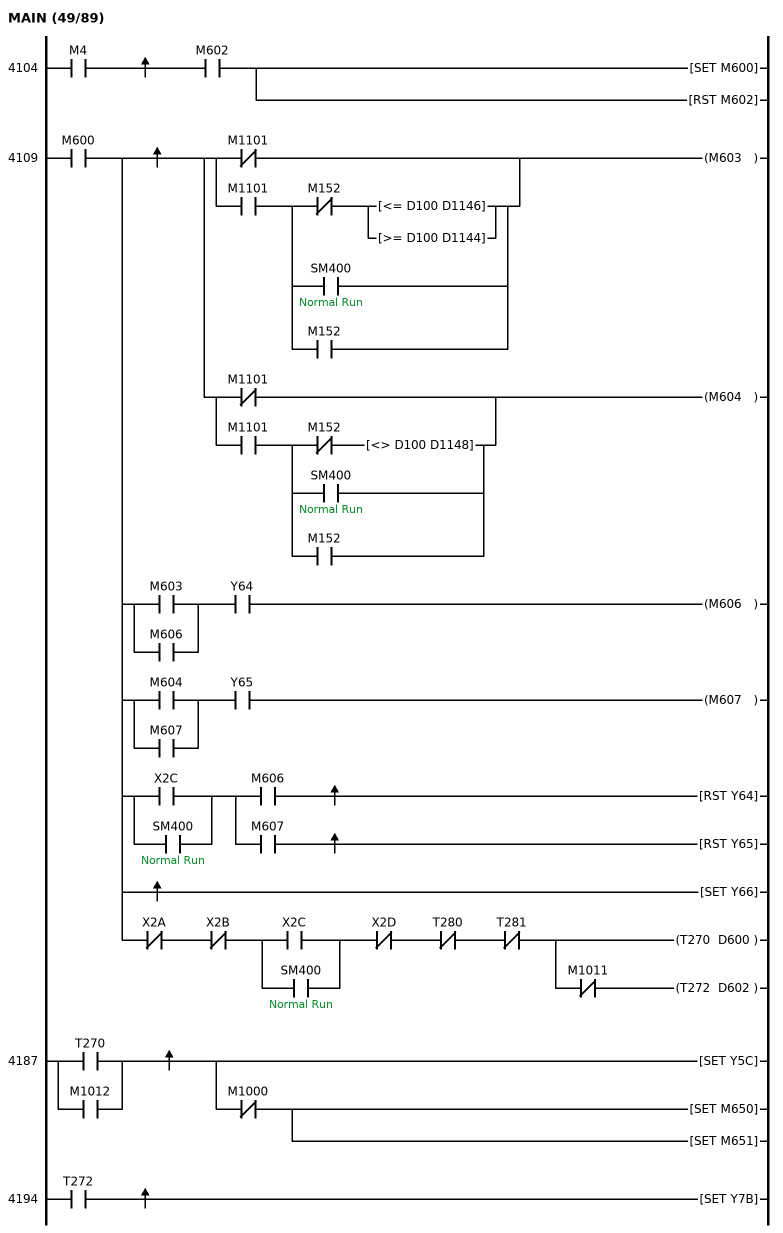
[picture p48: ladder of MAIN, rungs at steps 4104 to 4194]
4104  LD      M4
      MEP
      AND     M602
      SET     M600
      RST     M602
4109  LD      M600
      MPS
      MEP
      MPS
      LDI     M1101
      LD      M1101
      LDI     M152
      LD<=    D100 D1146
      OR>=    D100 D1144
      ANB
      OR      SM400  ; Normal Run
      OR      M152
      ANB
      ORB
      ANB
      OUT     M603
      MPP
      LDI     M1101
      LD      M1101
      LDI     M152
      AND<>   D100 D1148
      OR      SM400  ; Normal Run
      OR      M152
      ANB
      ORB
      ANB
      OUT     M604
      MRD
      LD      M603
      OR      M606
      ANB
      AND     Y64
      OUT     M606
      MRD
      LD      M604
      OR      M607
      ANB
      AND     Y65
      OUT     M607
      MRD
      LD      X2C
      OR      SM400  ; Normal Run
      ANB
      MPS
      AND     M606
      MEP
      RST     Y64
      MPP
      AND     M607
      MEP
      RST     Y65
      MRD
      MEP
      SET     Y66
      MPP
      ANI     X2A
      ANI     X2B
      LD      X2C
      OR      SM400  ; Normal Run
      ANB
      ANI     X2D
      ANI     T280
      ANI     T281
      OUT     T270 D600
      ANI     M1011
      OUT     T272 D602
4187  LD      T270
      OR      M1012
      MEP
      SET     Y5C
      ANI     M1000
      SET     M650
      SET     M651
4194  LD      T272
      MEP
      SET     Y7B
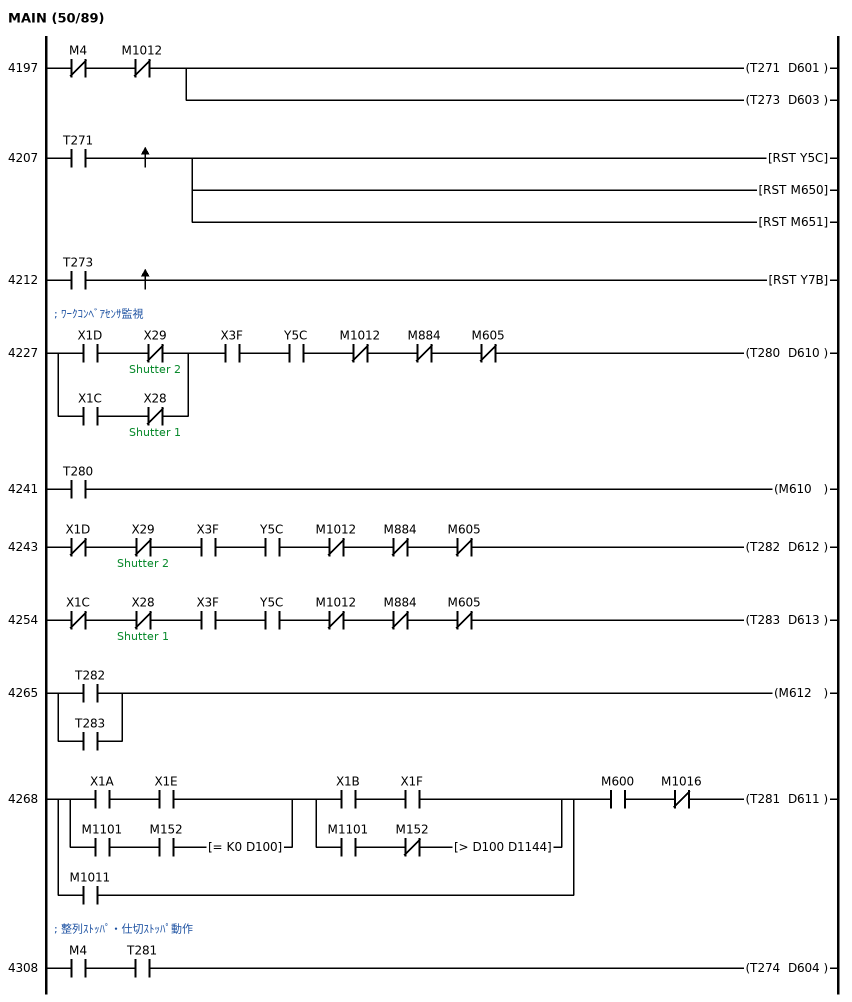
4197  LDI     M4
      ANI     M1012
      OUT     T271 D601
      OUT     T273 D603
4207  LD      T271
      MEP
      RST     Y5C
      RST     M650
      RST     M651
4212  LD      T273
      MEP
      RST     Y7B
; ﾜｰｸｺﾝﾍﾞｱｾﾝｻ監視
4227  LD      X1D
      ANI     X29  ; Shutter 2
      LD      X1C
      ANI     X28  ; Shutter 1
      ORB
      AND     X3F
      AND     Y5C
      ANI     M1012
      ANI     M884
      ANI     M605
      OUT     T280 D610
4241  LD      T280
      OUT     M610
4243  LDI     X1D
      ANI     X29  ; Shutter 2
      AND     X3F
      AND     Y5C
      ANI     M1012
      ANI     M884
      ANI     M605
      OUT     T282 D612
4254  LDI     X1C
      ANI     X28  ; Shutter 1
      AND     X3F
      AND     Y5C
      ANI     M1012
      ANI     M884
      ANI     M605
      OUT     T283 D613
4265  LD      T282
      OR      T283
      OUT     M612
4268  LD      X1A
      AND     X1E
      LD      M1101
      AND     M152
      AND=    K0 D100
      ORB
      LD      X1B
      AND     X1F
      LD      M1101
      ANI     M152
      AND>    D100 D1144
      ORB
      ANB
      OR      M1011
      AND     M600
      ANI     M1016
      OUT     T281 D611
; 整列ｽﾄｯﾊﾟ・仕切ｽﾄｯﾊﾟ動作
4308  LD      M4
      AND     T281
      OUT     T274 D604
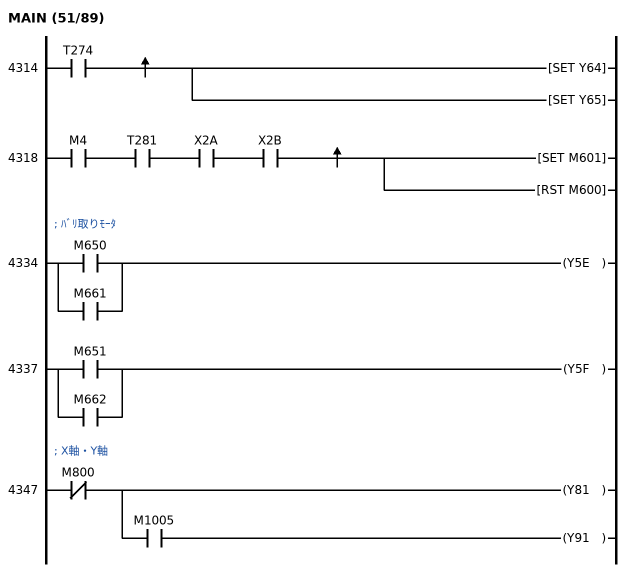
4314  LD      T274
      MEP
      SET     Y64
      SET     Y65
4318  LD      M4
      AND     T281
      AND     X2A
      AND     X2B
      MEP
      SET     M601
      RST     M600
; ﾊﾞﾘ取りﾓｰﾀ
4334  LD      M650
      OR      M661
      OUT     Y5E
4337  LD      M651
      OR      M662
      OUT     Y5F
; X軸・Y軸
; 
4347  LDI     M800
      OUT     Y81
      AND     M1005
      OUT     Y91
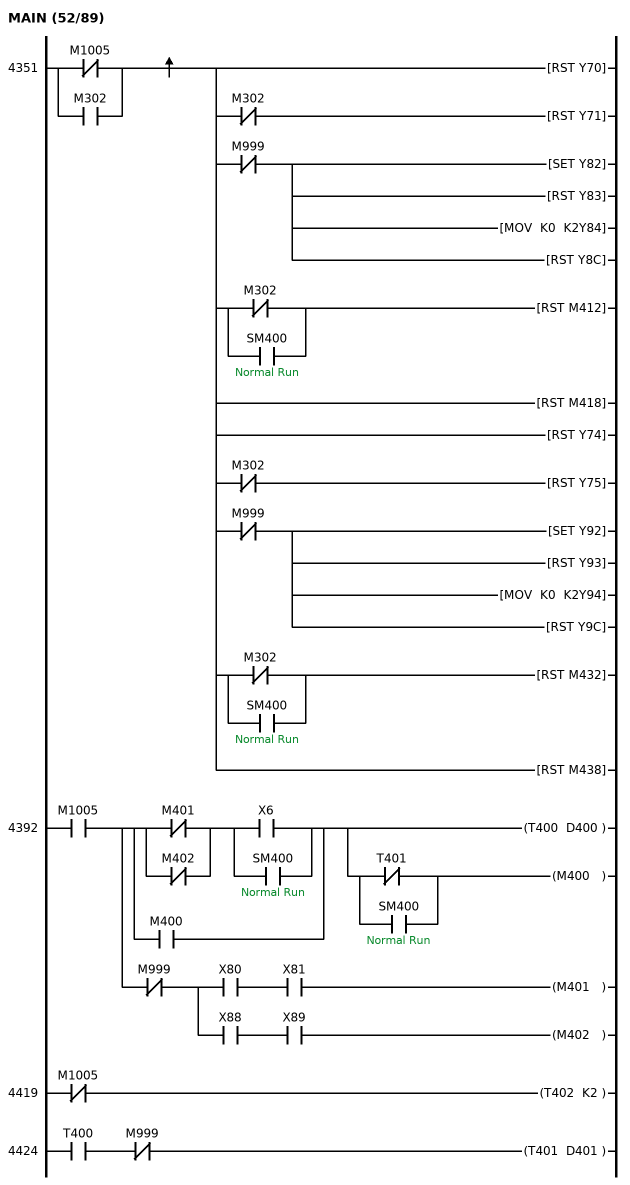
4351  LDI     M1005
      OR      M302
      MEP
      RST     Y70
      MPS
      ANI     M302
      RST     Y71
      MRD
      ANI     M999
      SET     Y82
      RST     Y83
      MOV     K0 K2Y84
      RST     Y8C
      MRD
      LDI     M302
      OR      SM400  ; Normal Run
      ANB
      RST     M412
      MPP
      RST     M418
      RST     Y74
      MPS
      ANI     M302
      RST     Y75
      MRD
      ANI     M999
      SET     Y92
      RST     Y93
      MOV     K0 K2Y94
      RST     Y9C
      MRD
      LDI     M302
      OR      SM400  ; Normal Run
      ANB
      RST     M432
      MPP
      RST     M438
4392  LD      M1005
      MPS
      LDI     M401
      ORI     M402
      LD      X6
      OR      SM400  ; Normal Run
      ANB
      OR      M400
      ANB
      OUT     T400 D400
      LDI     T401
      OR      SM400  ; Normal Run
      ANB
      OUT     M400
      MPP
      ANI     M999
      MPS
      AND     X80
      AND     X81
      OUT     M401
      MPP
      AND     X88
      AND     X89
      OUT     M402
4419  LDI     M1005
      OUT     T402 K2
4424  LD      T400
      ANI     M999
      OUT     T401 D401
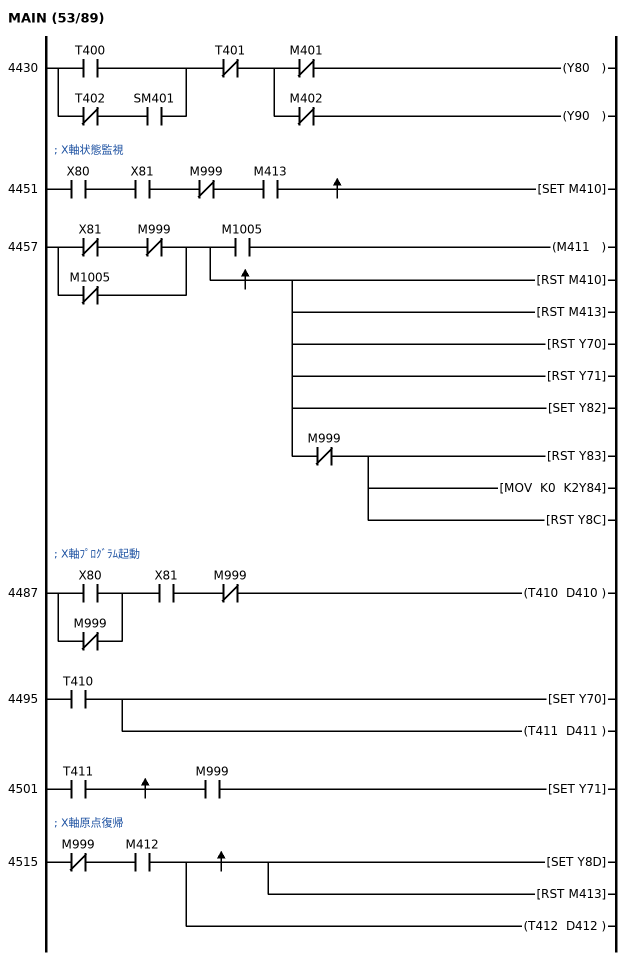
4430  LD      T400
      LDI     T402
      AND     SM401
      ORB
      ANI     T401
      MPS
      ANI     M401
      OUT     Y80
      MPP
      ANI     M402
      OUT     Y90
; X軸状態監視
4451  LD      X80
      AND     X81
      ANI     M999
      AND     M413
      MEP
      SET     M410
4457  LDI     X81
      ANI     M999
      ORI     M1005
      MPS
      AND     M1005
      OUT     M411
      MPP
      MEP
      RST     M410
      RST     M413
      RST     Y70
      RST     Y71
      SET     Y82
      ANI     M999
      RST     Y83
      MOV     K0 K2Y84
      RST     Y8C
; X軸ﾌﾟﾛｸﾞﾗﾑ起動
4487  LD      X80
      ORI     M999
      AND     X81
      ANI     M999
      OUT     T410 D410
4495  LD      T410
      SET     Y70
      OUT     T411 D411
4501  LD      T411
      MEP
      AND     M999
      SET     Y71
; X軸原点復帰
4515  LDI     M999
      AND     M412
      MPS
      MEP
      SET     Y8D
      RST     M413
      MPP
      OUT     T412 D412
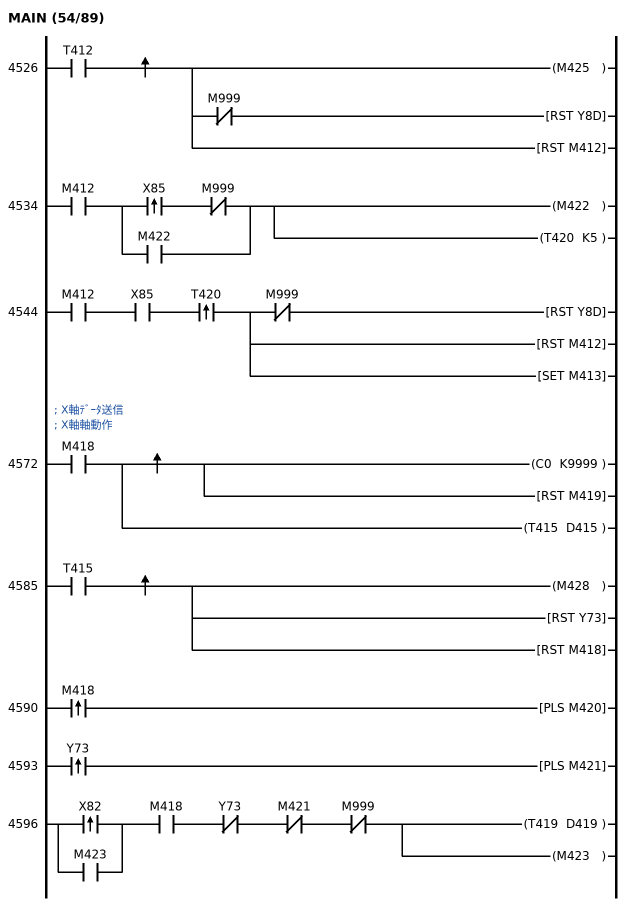
4526  LD      T412
      MEP
      OUT     M425
      MPS
      ANI     M999
      RST     Y8D
      MPP
      RST     M412
4534  LD      M412
      LDP     X85
      ANI     M999
      OR      M422
      ANB
      OUT     M422
      OUT     T420 K5
4544  LD      M412
      AND     X85
      ANDP    T420
      MPS
      ANI     M999
      RST     Y8D
      MPP
      RST     M412
      SET     M413
; X軸ﾃﾞｰﾀ送信
; X軸軸動作
4572  LD      M418
      MPS
      MEP
      OUT     C0 K9999
      RST     M419
      MPP
      OUT     T415 D415
4585  LD      T415
      MEP
      OUT     M428
      RST     Y73
      RST     M418
4590  LDP     M418
      PLS     M420
4593  LDP     Y73
      PLS     M421
4596  LDP     X82
      OR      M423
      AND     M418
      ANI     Y73
      ANI     M421
      ANI     M999
      OUT     T419 D419
      OUT     M423
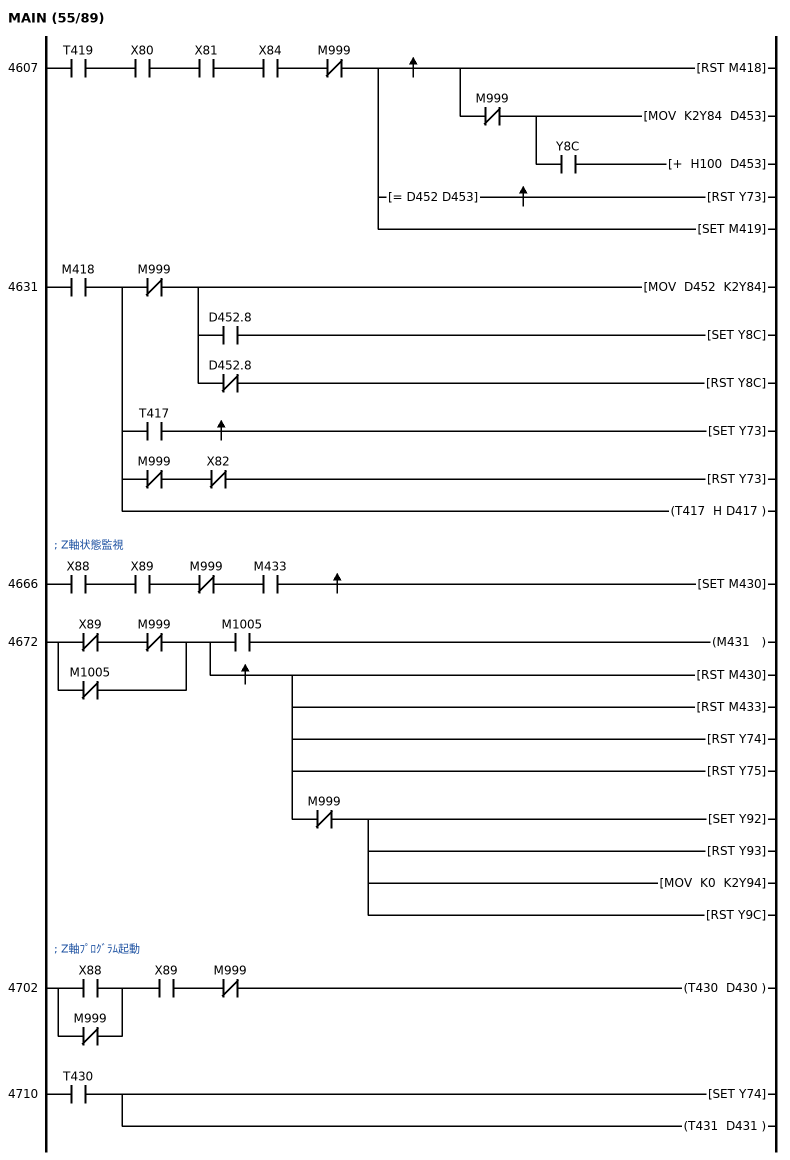
4607  LD      T419
      AND     X80
      AND     X81
      AND     X84
      ANI     M999
      MPS
      MEP
      RST     M418
      ANI     M999
      MOV     K2Y84 D453
      AND     Y8C
      +       H100 D453
      MRD
      AND=    D452 D453
      MEP
      RST     Y73
      MPP
      SET     M419
4631  LD      M418
      MPS
      ANI     M999
      MOV     D452 K2Y84
      MPS
      AND     D452.8
      SET     Y8C
      MPP
      ANI     D452.8
      RST     Y8C
      MRD
      AND     T417
      MEP
      SET     Y73
      MRD
      ANI     M999
      ANI     X82
      RST     Y73
      MPP
      OUTH    T417 D417
; Z軸状態監視
4666  LD      X88
      AND     X89
      ANI     M999
      AND     M433
      MEP
      SET     M430
4672  LDI     X89
      ANI     M999
      ORI     M1005
      MPS
      AND     M1005
      OUT     M431
      MPP
      MEP
      RST     M430
      RST     M433
      RST     Y74
      RST     Y75
      ANI     M999
      SET     Y92
      RST     Y93
      MOV     K0 K2Y94
      RST     Y9C
; Z軸ﾌﾟﾛｸﾞﾗﾑ起動
4702  LD      X88
      ORI     M999
      AND     X89
      ANI     M999
      OUT     T430 D430
4710  LD      T430
      SET     Y74
      OUT     T431 D431
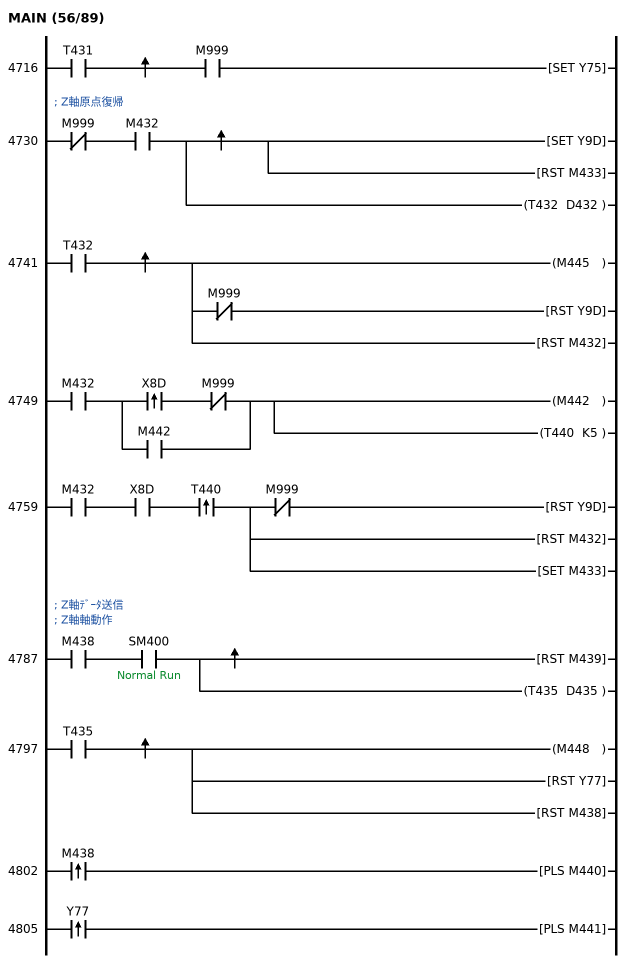
4716  LD      T431
      MEP
      AND     M999
      SET     Y75
; Z軸原点復帰
4730  LDI     M999
      AND     M432
      MPS
      MEP
      SET     Y9D
      RST     M433
      MPP
      OUT     T432 D432
4741  LD      T432
      MEP
      OUT     M445
      MPS
      ANI     M999
      RST     Y9D
      MPP
      RST     M432
4749  LD      M432
      LDP     X8D
      ANI     M999
      OR      M442
      ANB
      OUT     M442
      OUT     T440 K5
4759  LD      M432
      AND     X8D
      ANDP    T440
      MPS
      ANI     M999
      RST     Y9D
      MPP
      RST     M432
      SET     M433
; Z軸ﾃﾞｰﾀ送信
; Z軸軸動作
4787  LD      M438
      AND     SM400  ; Normal Run
      MPS
      MEP
      RST     M439
      MPP
      OUT     T435 D435
4797  LD      T435
      MEP
      OUT     M448
      RST     Y77
      RST     M438
4802  LDP     M438
      PLS     M440
4805  LDP     Y77
      PLS     M441
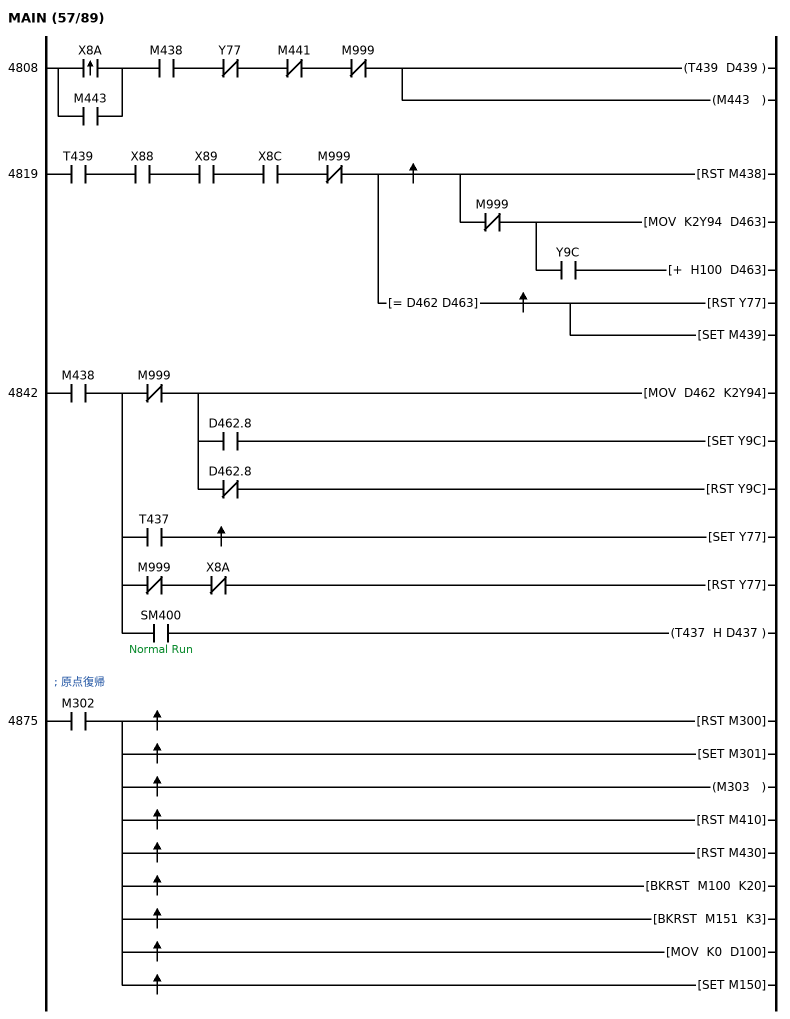
4808  LDP     X8A
      OR      M443
      AND     M438
      ANI     Y77
      ANI     M441
      ANI     M999
      OUT     T439 D439
      OUT     M443
4819  LD      T439
      AND     X88
      AND     X89
      AND     X8C
      ANI     M999
      MPS
      MEP
      RST     M438
      ANI     M999
      MOV     K2Y94 D463
      AND     Y9C
      +       H100 D463
      MPP
      AND=    D462 D463
      MEP
      RST     Y77
      SET     M439
4842  LD      M438
      MPS
      ANI     M999
      MOV     D462 K2Y94
      MPS
      AND     D462.8
      SET     Y9C
      MPP
      ANI     D462.8
      RST     Y9C
      MRD
      AND     T437
      MEP
      SET     Y77
      MRD
      ANI     M999
      ANI     X8A
      RST     Y77
      MPP
      AND     SM400  ; Normal Run
      OUTH    T437 D437
; 原点復帰
; 
4875  LD      M302
      MPS
      MEP
      RST     M300
      MRD
      MEP
      SET     M301
      MRD
      MEP
      OUT     M303
      MRD
      MEP
      RST     M410
      MRD
      MEP
      RST     M430
      MRD
      MEP
      BKRST   M100 K20
      MRD
      MEP
      BKRST   M151 K3
      MRD
      MEP
      MOV     K0 D100
      MPP
      MEP
      SET     M150
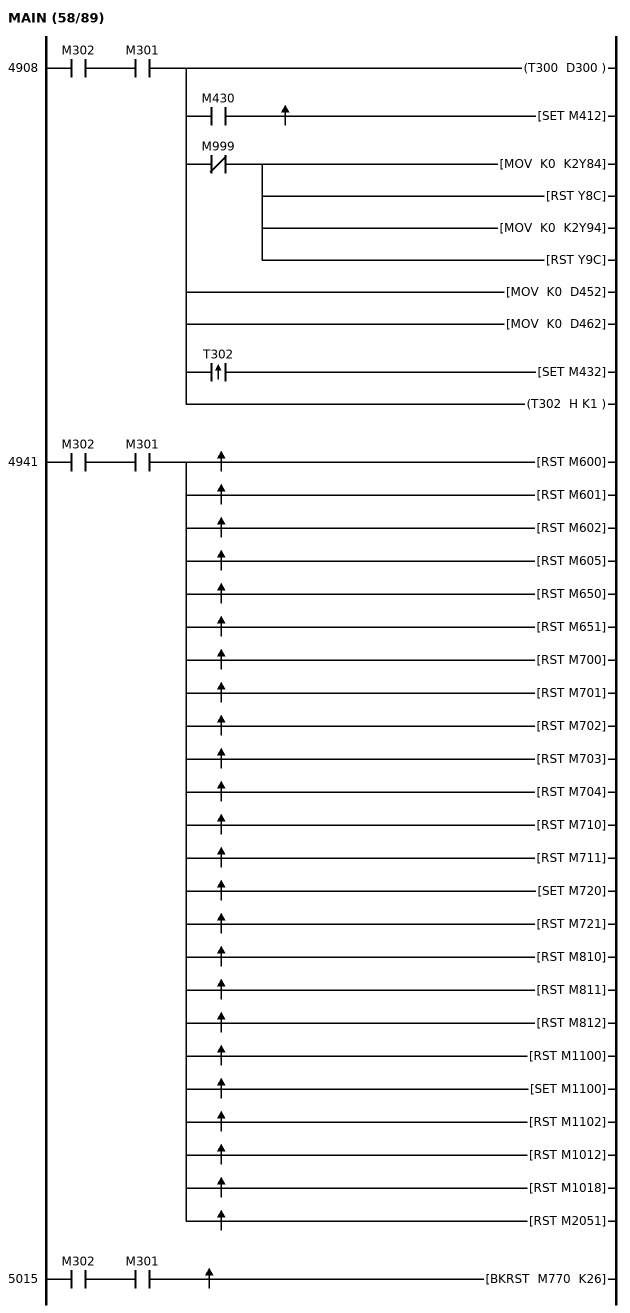
4908  LD      M302
      AND     M301
      OUT     T300 D300
      MPS
      AND     M430
      MEP
      SET     M412
      MRD
      ANI     M999
      MOV     K0 K2Y84
      RST     Y8C
      MOV     K0 K2Y94
      RST     Y9C
      MPP
      MOV     K0 D452
      MOV     K0 D462
      MPS
      ANDP    T302
      SET     M432
      MPP
      OUTH    T302 K1
4941  LD      M302
      AND     M301
      MPS
      MEP
      RST     M600
      MRD
      MEP
      RST     M601
      MRD
      MEP
      RST     M602
      MRD
      MEP
      RST     M605
      MRD
      MEP
      RST     M650
      MRD
      MEP
      RST     M651
      MRD
      MEP
      RST     M700
      MRD
      MEP
      RST     M701
      MRD
      MEP
      RST     M702
      MRD
      MEP
      RST     M703
      MRD
      MEP
      RST     M704
      MRD
      MEP
      RST     M710
      MRD
      MEP
      RST     M711
      MRD
      MEP
      SET     M720
      MRD
      MEP
      RST     M721
      MRD
      MEP
      RST     M810
      MRD
      MEP
      RST     M811
      MRD
      MEP
      RST     M812
      MRD
      MEP
      RST     M1100
      MRD
      MEP
      SET     M1100
      MRD
      MEP
      RST     M1102
      MRD
      MEP
      RST     M1012
      MRD
      MEP
      RST     M1018
      MPP
      MEP
      RST     M2051
5015  LD      M302
      AND     M301
      MEP
      BKRST   M770 K26
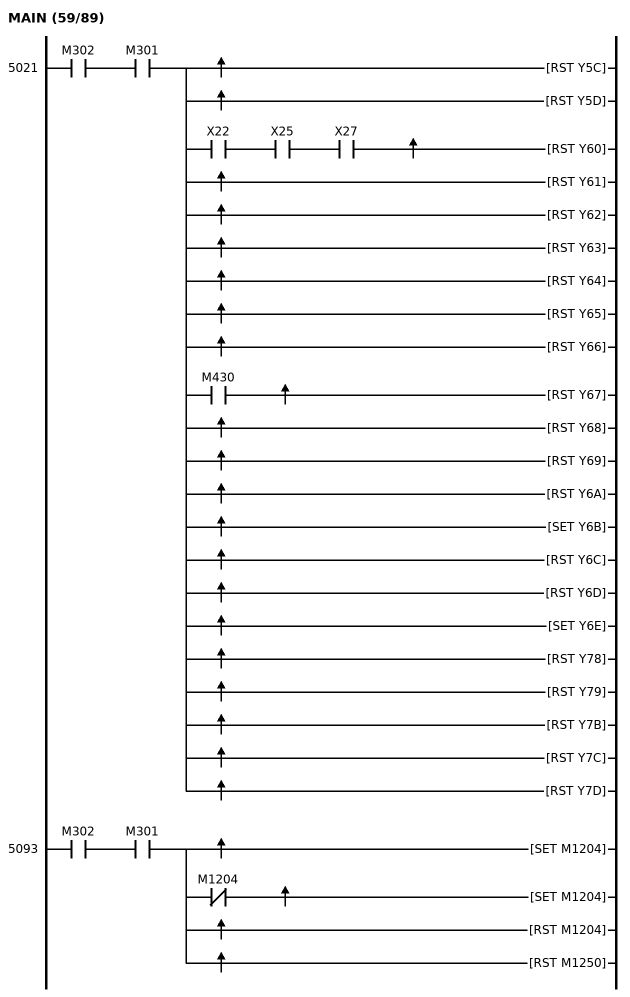
5021  LD      M302
      AND     M301
      MPS
      MEP
      RST     Y5C
      MRD
      MEP
      RST     Y5D
      MRD
      AND     X22
      AND     X25
      AND     X27
      MEP
      RST     Y60
      MRD
      MEP
      RST     Y61
      MRD
      MEP
      RST     Y62
      MRD
      MEP
      RST     Y63
      MRD
      MEP
      RST     Y64
      MRD
      MEP
      RST     Y65
      MRD
      MEP
      RST     Y66
      MRD
      AND     M430
      MEP
      RST     Y67
      MRD
      MEP
      RST     Y68
      MRD
      MEP
      RST     Y69
      MRD
      MEP
      RST     Y6A
      MRD
      MEP
      SET     Y6B
      MRD
      MEP
      RST     Y6C
      MRD
      MEP
      RST     Y6D
      MRD
      MEP
      SET     Y6E
      MRD
      MEP
      RST     Y78
      MRD
      MEP
      RST     Y79
      MRD
      MEP
      RST     Y7B
      MRD
      MEP
      RST     Y7C
      MPP
      MEP
      RST     Y7D
5093  LD      M302
      AND     M301
      MPS
      MEP
      SET     M1204
      MRD
      ANI     M1204
      MEP
      SET     M1204
      MRD
      MEP
      RST     M1204
      MPP
      MEP
      RST     M1250
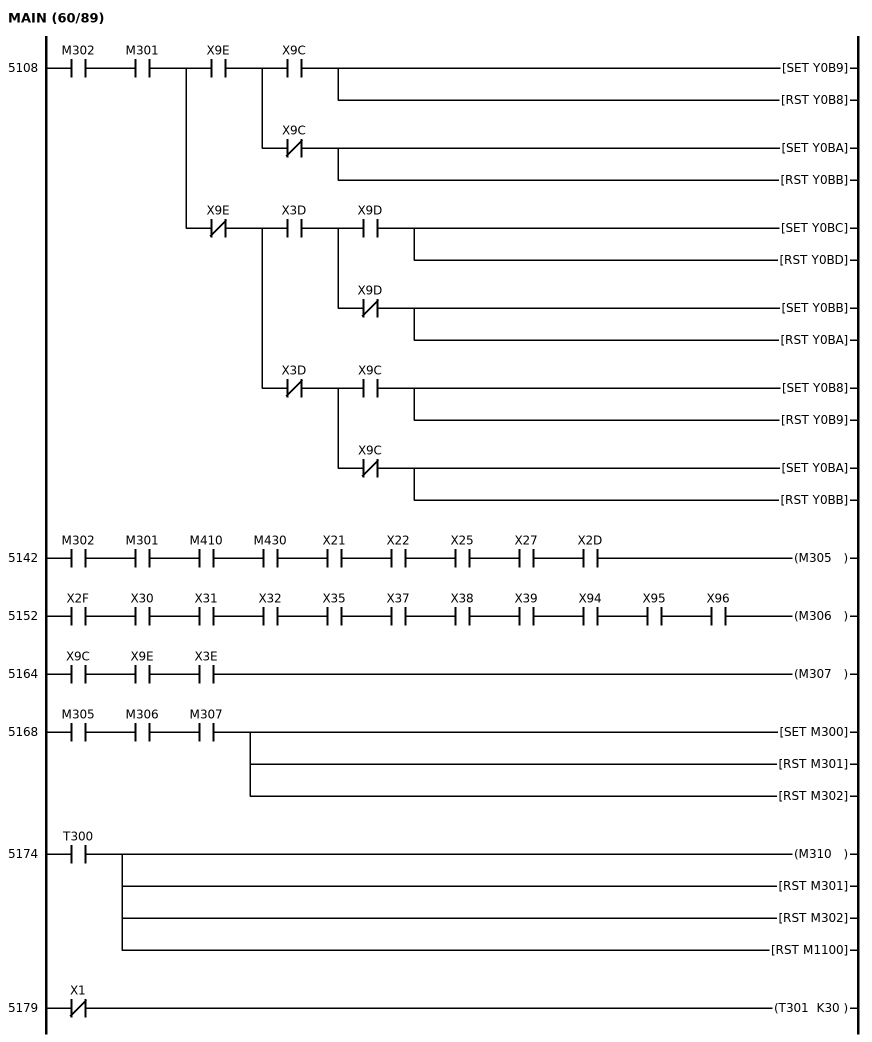
5108  LD      M302
      AND     M301
      MPS
      AND     X9E
      MPS
      AND     X9C
      SET     Y0B9
      RST     Y0B8
      MPP
      ANI     X9C
      SET     Y0BA
      RST     Y0BB
      MPP
      ANI     X9E
      MPS
      AND     X3D
      MPS
      AND     X9D
      SET     Y0BC
      RST     Y0BD
      MPP
      ANI     X9D
      SET     Y0BB
      RST     Y0BA
      MPP
      ANI     X3D
      MPS
      AND     X9C
      SET     Y0B8
      RST     Y0B9
      MPP
      ANI     X9C
      SET     Y0BA
      RST     Y0BB
5142  LD      M302
      AND     M301
      AND     M410
      AND     M430
      AND     X21
      AND     X22
      AND     X25
      AND     X27
      AND     X2D
      OUT     M305
5152  LD      X2F
      AND     X30
      AND     X31
      AND     X32
      AND     X35
      AND     X37
      AND     X38
      AND     X39
      AND     X94
      AND     X95
      AND     X96
      OUT     M306
5164  LD      X9C
      AND     X9E
      AND     X3E
      OUT     M307
5168  LD      M305
      AND     M306
      AND     M307
      SET     M300
      RST     M301
      RST     M302
5174  LD      T300
      OUT     M310
      RST     M301
      RST     M302
      RST     M1100
5179  LDI     X1
      OUT     T301 K30
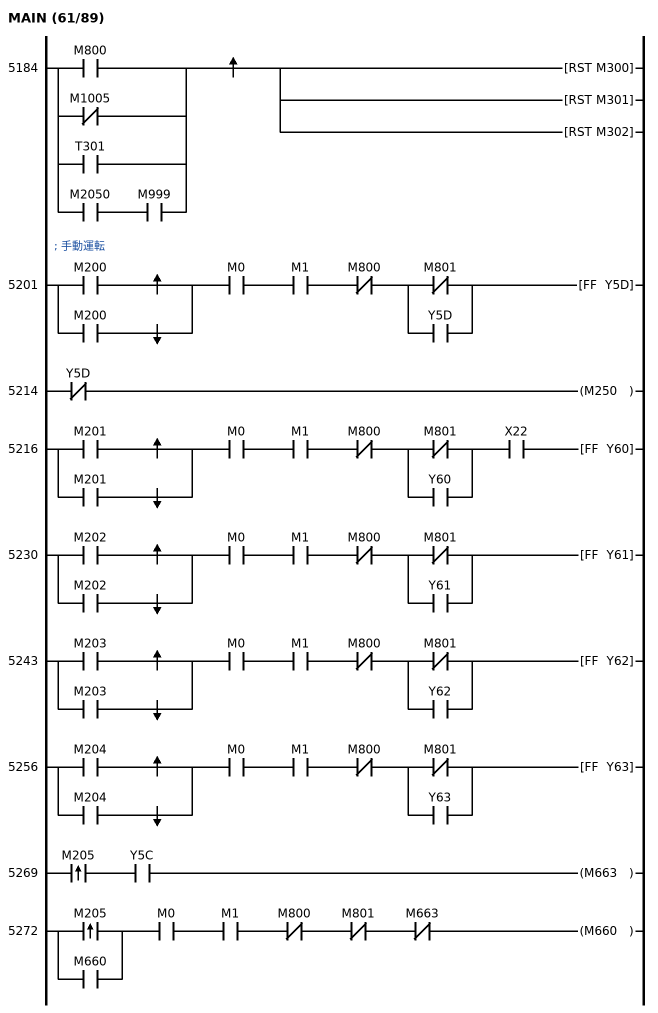
5184  LD      M800
      ORI     M1005
      OR      T301
      LD      M2050
      AND     M999
      ORB
      MEP
      RST     M300
      RST     M301
      RST     M302
; 手動運転
; 
5201  LD      M200
      MEP
      LD      M200
      MEF
      ORB
      AND     M0
      AND     M1
      ANI     M800
      LDI     M801
      OR      Y5D
      ANB
      FF      Y5D
5214  LDI     Y5D
      OUT     M250
5216  LD      M201
      MEP
      LD      M201
      MEF
      ORB
      AND     M0
      AND     M1
      ANI     M800
      LDI     M801
      OR      Y60
      ANB
      AND     X22
      FF      Y60
5230  LD      M202
      MEP
      LD      M202
      MEF
      ORB
      AND     M0
      AND     M1
      ANI     M800
      LDI     M801
      OR      Y61
      ANB
      FF      Y61
5243  LD      M203
      MEP
      LD      M203
      MEF
      ORB
      AND     M0
      AND     M1
      ANI     M800
      LDI     M801
      OR      Y62
      ANB
      FF      Y62
5256  LD      M204
      MEP
      LD      M204
      MEF
      ORB
      AND     M0
      AND     M1
      ANI     M800
      LDI     M801
      OR      Y63
      ANB
      FF      Y63
5269  LDP     M205
      AND     Y5C
      OUT     M663
5272  LDP     M205
      OR      M660
      AND     M0
      AND     M1
      ANI     M800
      ANI     M801
      ANI     M663
      OUT     M660
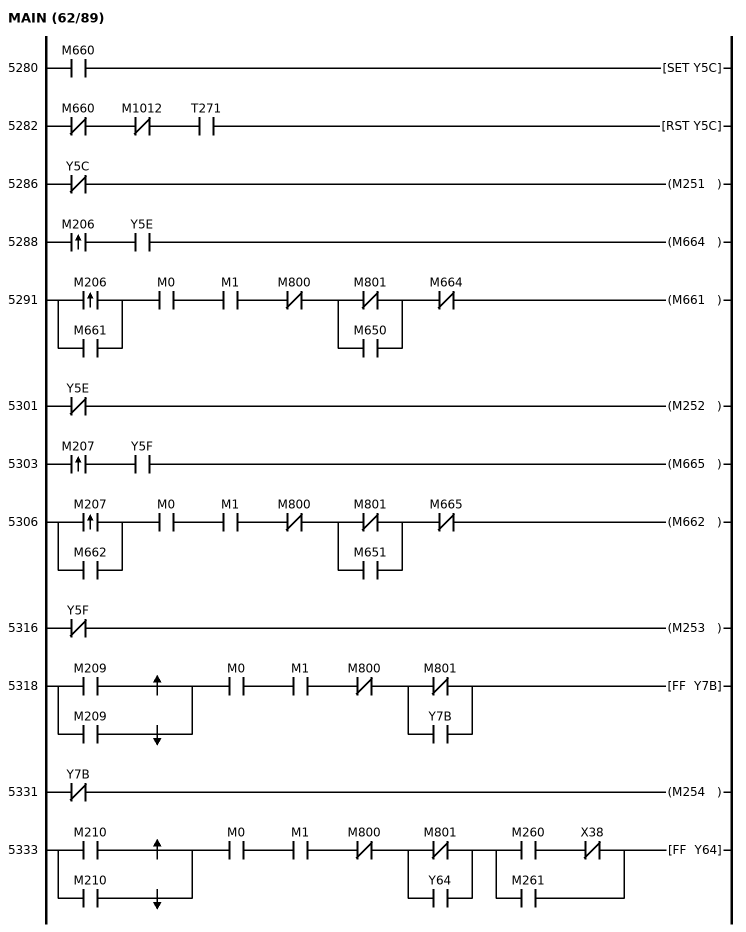
5280  LD      M660
      SET     Y5C
5282  LDI     M660
      ANI     M1012
      AND     T271
      RST     Y5C
5286  LDI     Y5C
      OUT     M251
5288  LDP     M206
      AND     Y5E
      OUT     M664
5291  LDP     M206
      OR      M661
      AND     M0
      AND     M1
      ANI     M800
      LDI     M801
      OR      M650
      ANB
      ANI     M664
      OUT     M661
5301  LDI     Y5E
      OUT     M252
5303  LDP     M207
      AND     Y5F
      OUT     M665
5306  LDP     M207
      OR      M662
      AND     M0
      AND     M1
      ANI     M800
      LDI     M801
      OR      M651
      ANB
      ANI     M665
      OUT     M662
5316  LDI     Y5F
      OUT     M253
5318  LD      M209
      MEP
      LD      M209
      MEF
      ORB
      AND     M0
      AND     M1
      ANI     M800
      LDI     M801
      OR      Y7B
      ANB
      FF      Y7B
5331  LDI     Y7B
      OUT     M254
5333  LD      M210
      MEP
      LD      M210
      MEF
      ORB
      AND     M0
      AND     M1
      ANI     M800
      LDI     M801
      OR      Y64
      ANB
      LD      M260
      ANI     X38
      OR      M261
      ANB
      FF      Y64
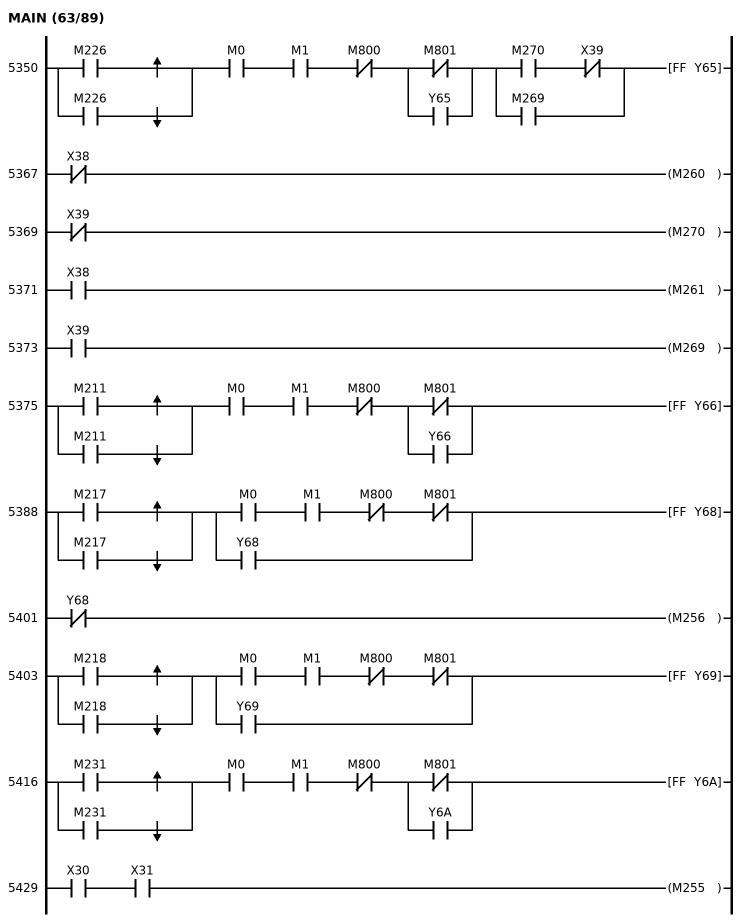
5350  LD      M226
      MEP
      LD      M226
      MEF
      ORB
      AND     M0
      AND     M1
      ANI     M800
      LDI     M801
      OR      Y65
      ANB
      LD      M270
      ANI     X39
      OR      M269
      ANB
      FF      Y65
5367  LDI     X38
      OUT     M260
5369  LDI     X39
      OUT     M270
5371  LD      X38
      OUT     M261
5373  LD      X39
      OUT     M269
5375  LD      M211
      MEP
      LD      M211
      MEF
      ORB
      AND     M0
      AND     M1
      ANI     M800
      LDI     M801
      OR      Y66
      ANB
      FF      Y66
5388  LD      M217
      MEP
      LD      M217
      MEF
      ORB
      LD      M0
      AND     M1
      ANI     M800
      ANI     M801
      OR      Y68
      ANB
      FF      Y68
5401  LDI     Y68
      OUT     M256
5403  LD      M218
      MEP
      LD      M218
      MEF
      ORB
      LD      M0
      AND     M1
      ANI     M800
      ANI     M801
      OR      Y69
      ANB
      FF      Y69
5416  LD      M231
      MEP
      LD      M231
      MEF
      ORB
      AND     M0
      AND     M1
      ANI     M800
      LDI     M801
      OR      Y6A
      ANB
      FF      Y6A
5429  LD      X30
      AND     X31
      OUT     M255
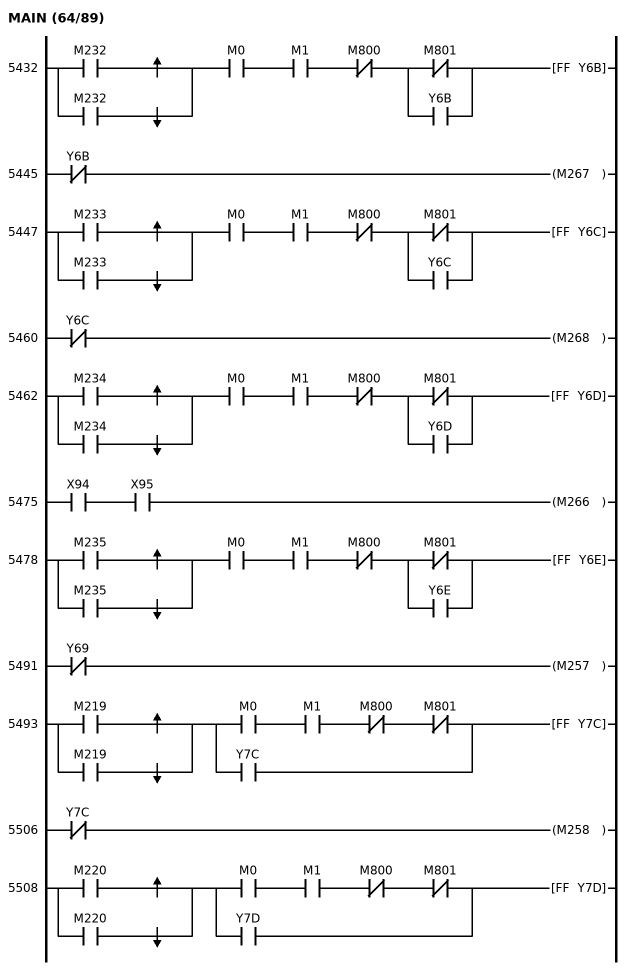
5432  LD      M232
      MEP
      LD      M232
      MEF
      ORB
      AND     M0
      AND     M1
      ANI     M800
      LDI     M801
      OR      Y6B
      ANB
      FF      Y6B
5445  LDI     Y6B
      OUT     M267
5447  LD      M233
      MEP
      LD      M233
      MEF
      ORB
      AND     M0
      AND     M1
      ANI     M800
      LDI     M801
      OR      Y6C
      ANB
      FF      Y6C
5460  LDI     Y6C
      OUT     M268
5462  LD      M234
      MEP
      LD      M234
      MEF
      ORB
      AND     M0
      AND     M1
      ANI     M800
      LDI     M801
      OR      Y6D
      ANB
      FF      Y6D
5475  LD      X94
      AND     X95
      OUT     M266
5478  LD      M235
      MEP
      LD      M235
      MEF
      ORB
      AND     M0
      AND     M1
      ANI     M800
      LDI     M801
      OR      Y6E
      ANB
      FF      Y6E
5491  LDI     Y69
      OUT     M257
5493  LD      M219
      MEP
      LD      M219
      MEF
      ORB
      LD      M0
      AND     M1
      ANI     M800
      ANI     M801
      OR      Y7C
      ANB
      FF      Y7C
5506  LDI     Y7C
      OUT     M258
5508  LD      M220
      MEP
      LD      M220
      MEF
      ORB
      LD      M0
      AND     M1
      ANI     M800
      ANI     M801
      OR      Y7D
      ANB
      FF      Y7D
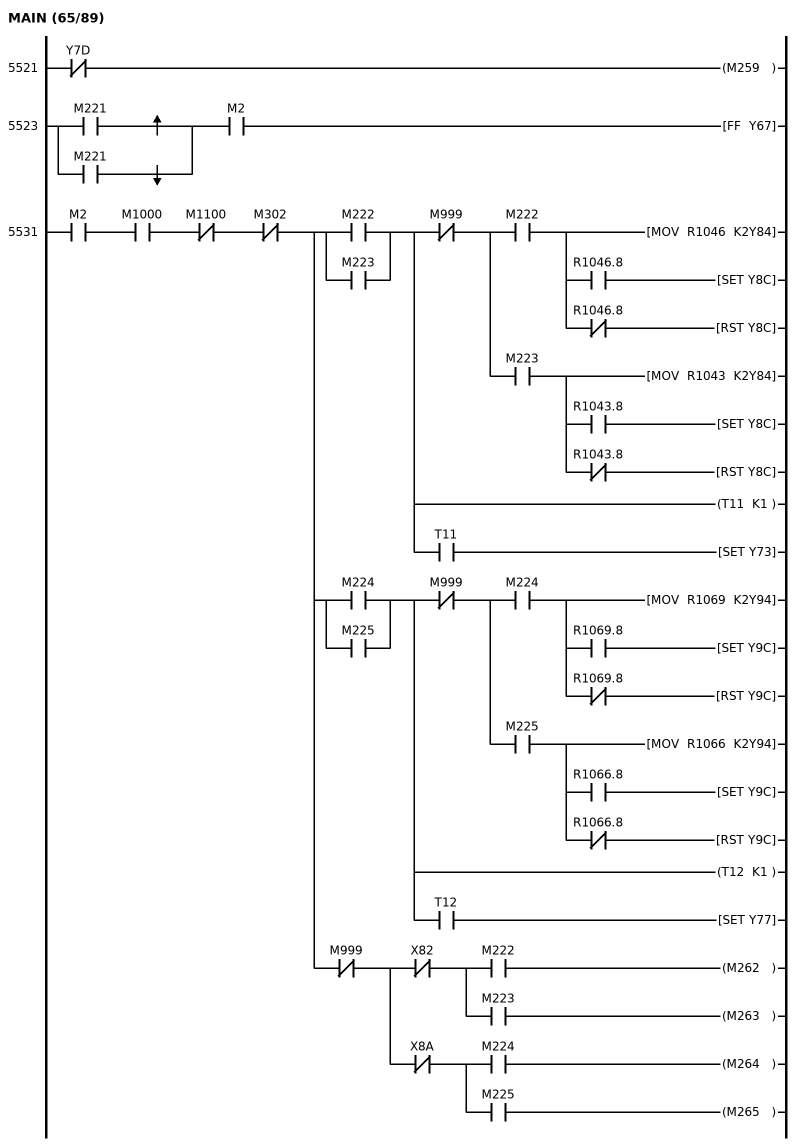
5521  LDI     Y7D
      OUT     M259
5523  LD      M221
      MEP
      LD      M221
      MEF
      ORB
      AND     M2
      FF      Y67
5531  LD      M2
      AND     M1000
      ANI     M1100
      ANI     M302
      MPS
      LD      M222
      OR      M223
      ANB
      MPS
      ANI     M999
      MPS
      AND     M222
      MOV     R1046 K2Y84
      MPS
      AND     R1046.8
      SET     Y8C
      MPP
      ANI     R1046.8
      RST     Y8C
      MPP
      AND     M223
      MOV     R1043 K2Y84
      MPS
      AND     R1043.8
      SET     Y8C
      MPP
      ANI     R1043.8
      RST     Y8C
      MPP
      OUT     T11 K1
      AND     T11
      SET     Y73
      MRD
      LD      M224
      OR      M225
      ANB
      MPS
      ANI     M999
      MPS
      AND     M224
      MOV     R1069 K2Y94
      MPS
      AND     R1069.8
      SET     Y9C
      MPP
      ANI     R1069.8
      RST     Y9C
      MPP
      AND     M225
      MOV     R1066 K2Y94
      MPS
      AND     R1066.8
      SET     Y9C
      MPP
      ANI     R1066.8
      RST     Y9C
      MPP
      OUT     T12 K1
      AND     T12
      SET     Y77
      MPP
      ANI     M999
      MPS
      ANI     X82
      MPS
      AND     M222
      OUT     M262
      MPP
      AND     M223
      OUT     M263
      MPP
      ANI     X8A
      MPS
      AND     M224
      OUT     M264
      MPP
      AND     M225
      OUT     M265
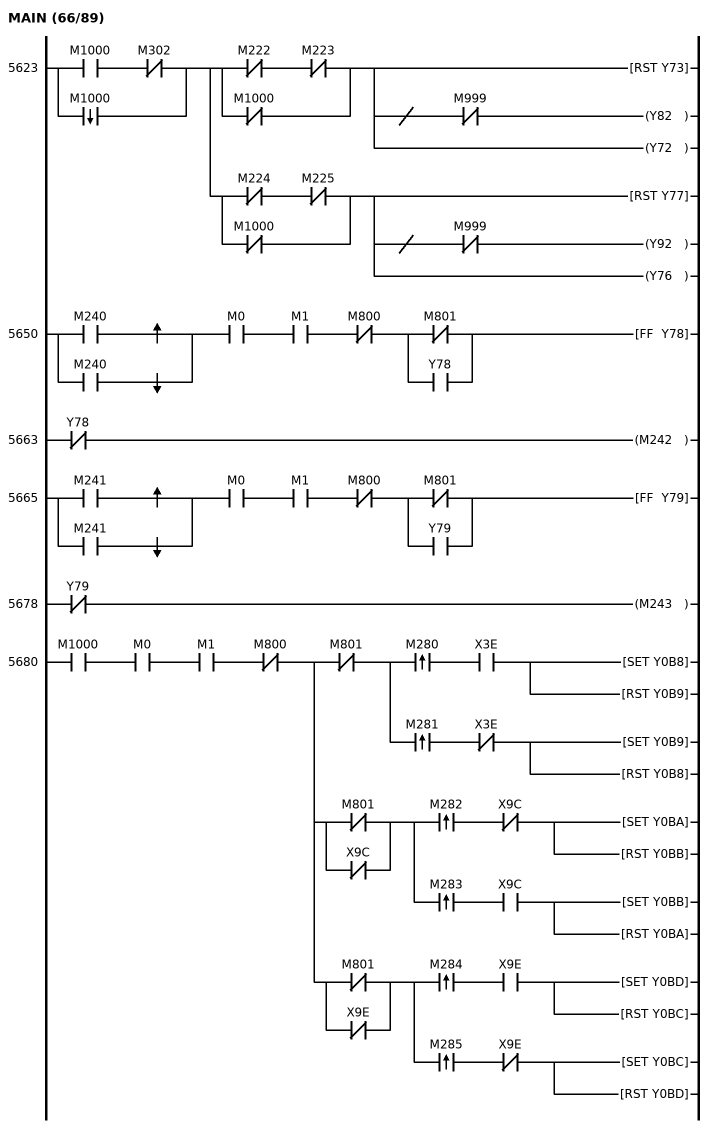
5623  LD      M1000
      ANI     M302
      ORF     M1000
      MPS
      LDI     M222
      ANI     M223
      ORI     M1000
      ANB
      RST     Y73
      MPS
      INV
      ANI     M999
      OUT     Y82
      MPP
      OUT     Y72
      MPP
      LDI     M224
      ANI     M225
      ORI     M1000
      ANB
      RST     Y77
      MPS
      INV
      ANI     M999
      OUT     Y92
      MPP
      OUT     Y76
5650  LD      M240
      MEP
      LD      M240
      MEF
      ORB
      AND     M0
      AND     M1
      ANI     M800
      LDI     M801
      OR      Y78
      ANB
      FF      Y78
5663  LDI     Y78
      OUT     M242
5665  LD      M241
      MEP
      LD      M241
      MEF
      ORB
      AND     M0
      AND     M1
      ANI     M800
      LDI     M801
      OR      Y79
      ANB
      FF      Y79
5678  LDI     Y79
      OUT     M243
5680  LD      M1000
      AND     M0
      AND     M1
      ANI     M800
      MPS
      ANI     M801
      MPS
      ANDP    M280
      AND     X3E
      SET     Y0B8
      RST     Y0B9
      MPP
      ANDP    M281
      ANI     X3E
      SET     Y0B9
      RST     Y0B8
      MRD
      LDI     M801
      ORI     X9C
      ANB
      MPS
      ANDP    M282
      ANI     X9C
      SET     Y0BA
      RST     Y0BB
      MPP
      ANDP    M283
      AND     X9C
      SET     Y0BB
      RST     Y0BA
      MPP
      LDI     M801
      ORI     X9E
      ANB
      MPS
      ANDP    M284
      AND     X9E
      SET     Y0BD
      RST     Y0BC
      MPP
      ANDP    M285
      ANI     X9E
      SET     Y0BC
      RST     Y0BD
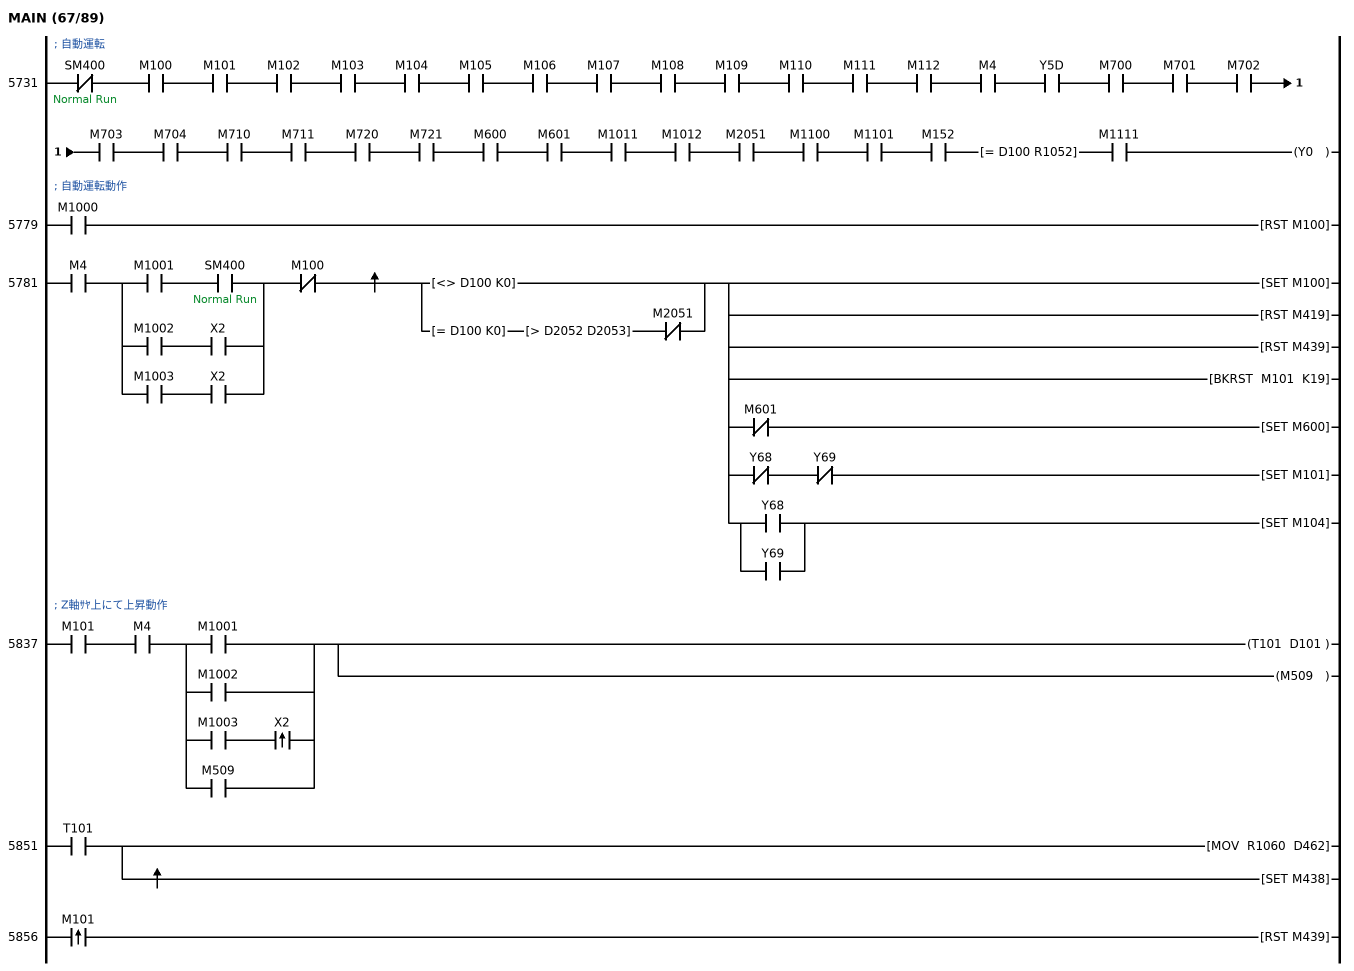
; 自動運転
; 
5731  LDI     SM400  ; Normal Run
      AND     M100
      AND     M101
      AND     M102
      AND     M103
      AND     M104
      AND     M105
      AND     M106
      AND     M107
      AND     M108
      AND     M109
      AND     M110
      AND     M111
      AND     M112
      AND     M4
      AND     Y5D
      AND     M700
      AND     M701
      AND     M702
      AND     M703
      AND     M704
      AND     M710
      AND     M711
      AND     M720
      AND     M721
      AND     M600
      AND     M601
      AND     M1011
      AND     M1012
      AND     M2051
      AND     M1100
      AND     M1101
      AND     M152
      AND=    D100 R1052
      AND     M1111
      OUT     Y0
; 自動運転動作
5779  LD      M1000
      RST     M100
5781  LD      M4
      LD      M1001
      AND     SM400  ; Normal Run
      LD      M1002
      AND     X2
      ORB
      LD      M1003
      AND     X2
      ORB
      ANB
      ANI     M100
      MEP
      LD<>    D100 K0
      LD=     D100 K0
      AND>    D2052 D2053
      ANI     M2051
      ORB
      ANB
      SET     M100
      RST     M419
      RST     M439
      BKRST   M101 K19
      MPS
      ANI     M601
      SET     M600
      MRD
      ANI     Y68
      ANI     Y69
      SET     M101
      MPP
      LD      Y68
      OR      Y69
      ANB
      SET     M104
; Z軸ｻﾔ上にて上昇動作
5837  LD      M101
      AND     M4
      LD      M1001
      OR      M1002
      LD      M1003
      ANDP    X2
      ORB
      OR      M509
      ANB
      OUT     T101 D101
      OUT     M509
5851  LD      T101
      MOV     R1060 D462
      MEP
      SET     M438
5856  LDP     M101
      RST     M439
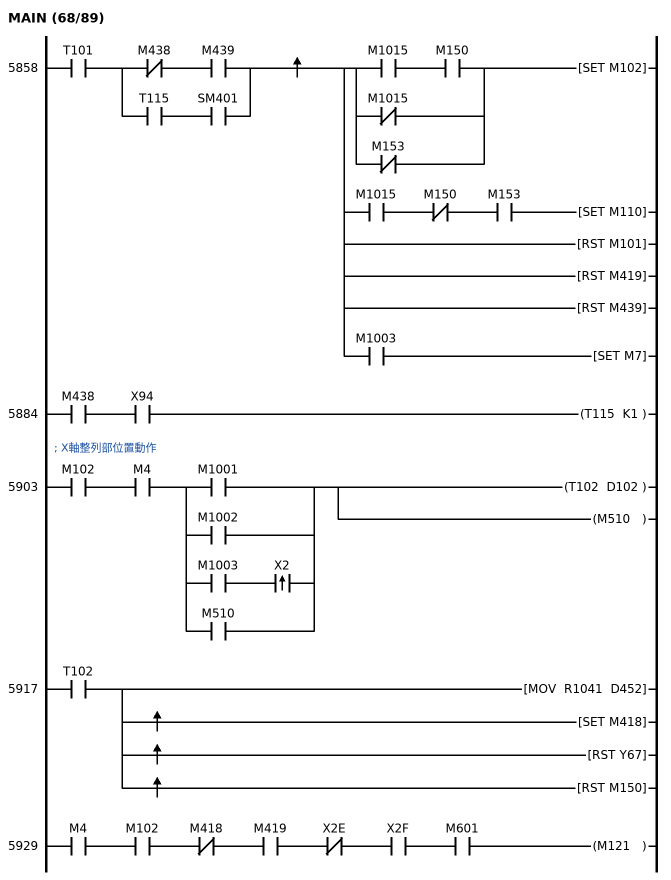
5858  LD      T101
      LDI     M438
      AND     M439
      LD      T115
      AND     SM401
      ORB
      ANB
      MEP
      MPS
      LD      M1015
      AND     M150
      ORI     M1015
      ORI     M153
      ANB
      SET     M102
      MRD
      AND     M1015
      ANI     M150
      AND     M153
      SET     M110
      MPP
      RST     M101
      RST     M419
      RST     M439
      AND     M1003
      SET     M7
5884  LD      M438
      AND     X94
      OUT     T115 K1
; X軸整列部位置動作
5903  LD      M102
      AND     M4
      LD      M1001
      OR      M1002
      LD      M1003
      ANDP    X2
      ORB
      OR      M510
      ANB
      OUT     T102 D102
      OUT     M510
5917  LD      T102
      MOV     R1041 D452
      MPS
      MEP
      SET     M418
      MRD
      MEP
      RST     Y67
      MPP
      MEP
      RST     M150
5929  LD      M4
      AND     M102
      ANI     M418
      AND     M419
      ANI     X2E
      AND     X2F
      AND     M601
      OUT     M121
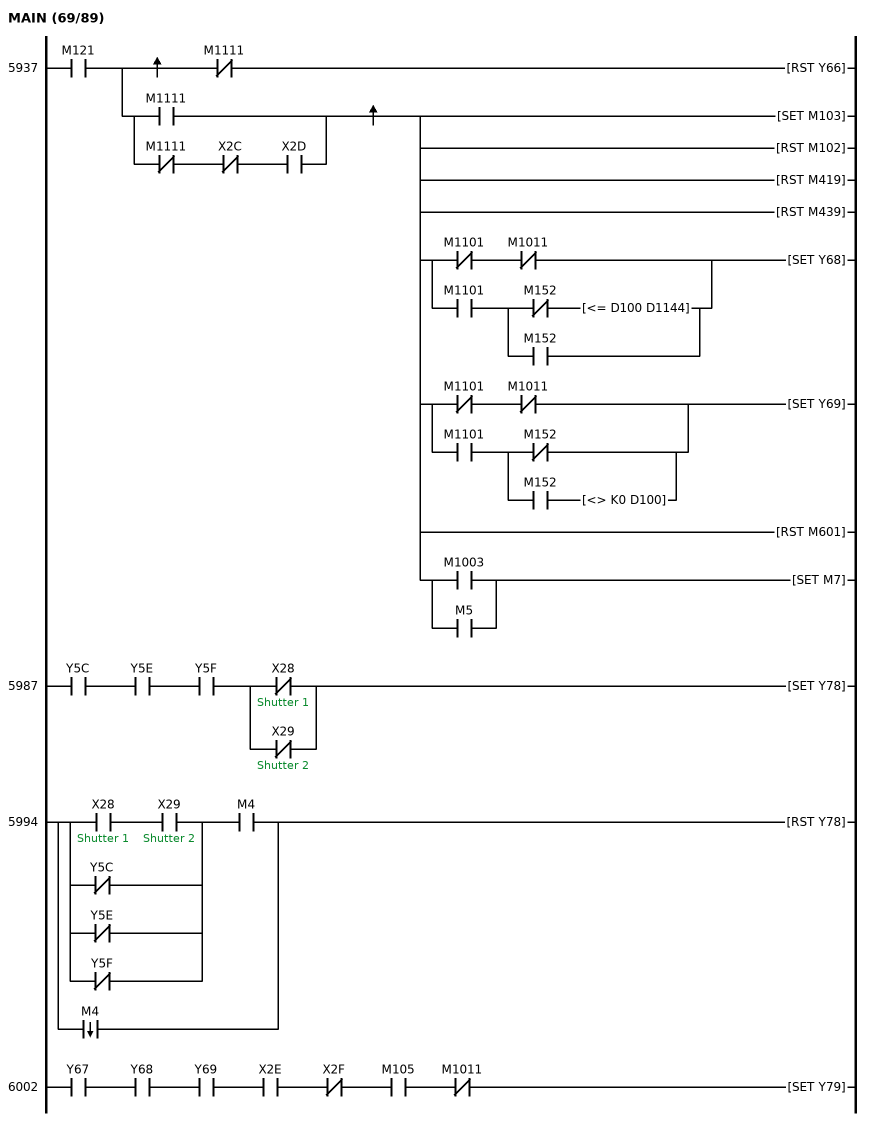
5937  LD      M121
      MPS
      MEP
      ANI     M1111
      RST     Y66
      MPP
      LD      M1111
      LDI     M1111
      ANI     X2C
      AND     X2D
      ORB
      ANB
      MEP
      SET     M103
      RST     M102
      RST     M419
      RST     M439
      MPS
      LDI     M1101
      ANI     M1011
      LD      M1101
      LDI     M152
      AND<=   D100 D1144
      OR      M152
      ANB
      ORB
      ANB
      SET     Y68
      MRD
      LDI     M1101
      ANI     M1011
      LD      M1101
      LDI     M152
      LD      M152
      AND<>   K0 D100
      ORB
      ANB
      ORB
      ANB
      SET     Y69
      MPP
      RST     M601
      LD      M1003
      OR      M5
      ANB
      SET     M7
5987  LD      Y5C
      AND     Y5E
      AND     Y5F
      LDI     X28  ; Shutter 1
      ORI     X29  ; Shutter 2
      ANB
      SET     Y78
5994  LD      X28  ; Shutter 1
      AND     X29  ; Shutter 2
      ORI     Y5C
      ORI     Y5E
      ORI     Y5F
      AND     M4
      ORF     M4
      RST     Y78
6002  LD      Y67
      AND     Y68
      AND     Y69
      AND     X2E
      ANI     X2F
      AND     M105
      ANI     M1011
      SET     Y79
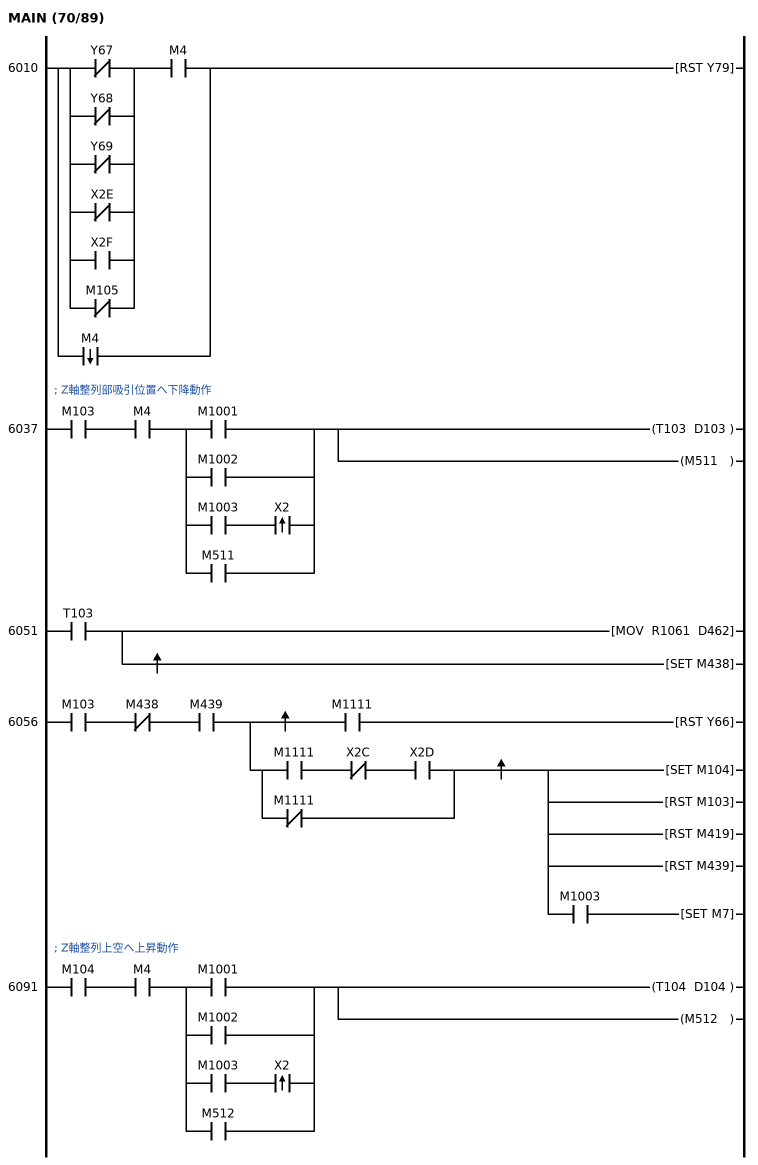
6010  LDI     Y67
      ORI     Y68
      ORI     Y69
      ORI     X2E
      OR      X2F
      ORI     M105
      AND     M4
      ORF     M4
      RST     Y79
; Z軸整列部吸引位置へ下降動作
6037  LD      M103
      AND     M4
      LD      M1001
      OR      M1002
      LD      M1003
      ANDP    X2
      ORB
      OR      M511
      ANB
      OUT     T103 D103
      OUT     M511
6051  LD      T103
      MOV     R1061 D462
      MEP
      SET     M438
6056  LD      M103
      ANI     M438
      AND     M439
      MPS
      MEP
      AND     M1111
      RST     Y66
      MPP
      LD      M1111
      ANI     X2C
      AND     X2D
      ORI     M1111
      ANB
      MEP
      SET     M104
      RST     M103
      RST     M419
      RST     M439
      AND     M1003
      SET     M7
; Z軸整列上空へ上昇動作
6091  LD      M104
      AND     M4
      LD      M1001
      OR      M1002
      LD      M1003
      ANDP    X2
      ORB
      OR      M512
      ANB
      OUT     T104 D104
      OUT     M512
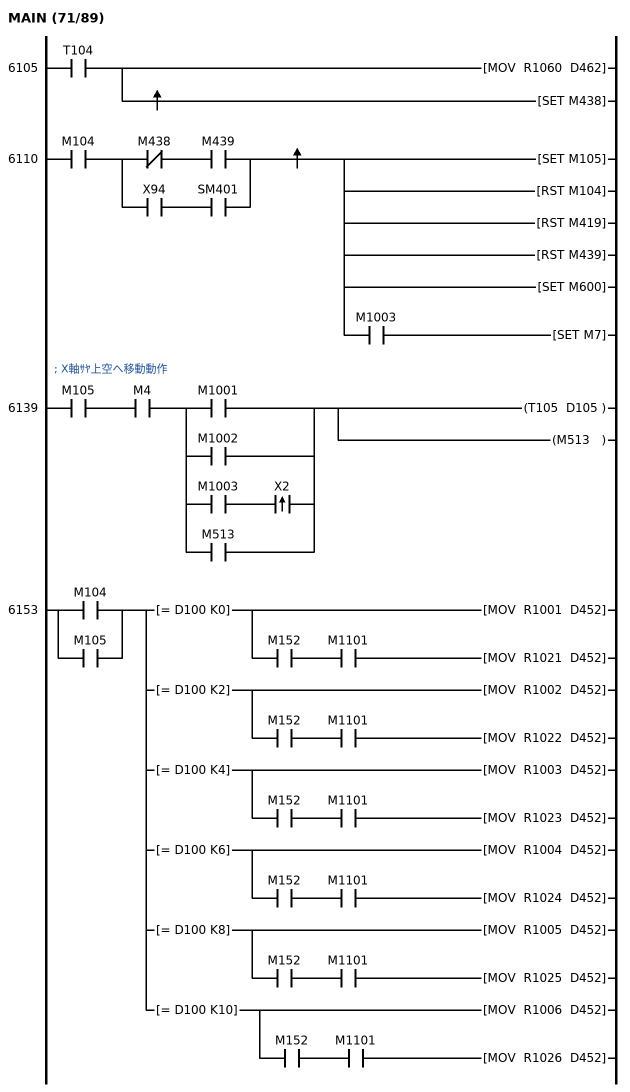
6105  LD      T104
      MOV     R1060 D462
      MEP
      SET     M438
6110  LD      M104
      LDI     M438
      AND     M439
      LD      X94
      AND     SM401
      ORB
      ANB
      MEP
      SET     M105
      RST     M104
      RST     M419
      RST     M439
      SET     M600
      AND     M1003
      SET     M7
; X軸ｻﾔ上空へ移動動作
6139  LD      M105
      AND     M4
      LD      M1001
      OR      M1002
      LD      M1003
      ANDP    X2
      ORB
      OR      M513
      ANB
      OUT     T105 D105
      OUT     M513
6153  LD      M104
      OR      M105
      MPS
      AND=    D100 K0
      MOV     R1001 D452
      AND     M152
      AND     M1101
      MOV     R1021 D452
      MRD
      AND=    D100 K2
      MOV     R1002 D452
      AND     M152
      AND     M1101
      MOV     R1022 D452
      MRD
      AND=    D100 K4
      MOV     R1003 D452
      AND     M152
      AND     M1101
      MOV     R1023 D452
      MRD
      AND=    D100 K6
      MOV     R1004 D452
      AND     M152
      AND     M1101
      MOV     R1024 D452
      MRD
      AND=    D100 K8
      MOV     R1005 D452
      AND     M152
      AND     M1101
      MOV     R1025 D452
      MPP
      AND=    D100 K10
      MOV     R1006 D452
      AND     M152
      AND     M1101
      MOV     R1026 D452
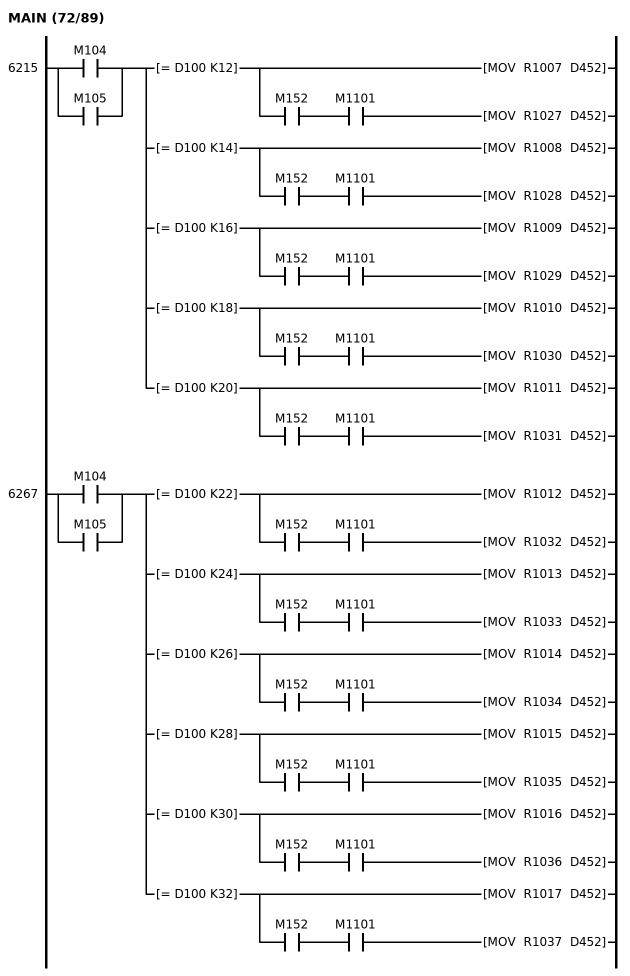
6215  LD      M104
      OR      M105
      MPS
      AND=    D100 K12
      MOV     R1007 D452
      AND     M152
      AND     M1101
      MOV     R1027 D452
      MRD
      AND=    D100 K14
      MOV     R1008 D452
      AND     M152
      AND     M1101
      MOV     R1028 D452
      MRD
      AND=    D100 K16
      MOV     R1009 D452
      AND     M152
      AND     M1101
      MOV     R1029 D452
      MRD
      AND=    D100 K18
      MOV     R1010 D452
      AND     M152
      AND     M1101
      MOV     R1030 D452
      MPP
      AND=    D100 K20
      MOV     R1011 D452
      AND     M152
      AND     M1101
      MOV     R1031 D452
6267  LD      M104
      OR      M105
      MPS
      AND=    D100 K22
      MOV     R1012 D452
      AND     M152
      AND     M1101
      MOV     R1032 D452
      MRD
      AND=    D100 K24
      MOV     R1013 D452
      AND     M152
      AND     M1101
      MOV     R1033 D452
      MRD
      AND=    D100 K26
      MOV     R1014 D452
      AND     M152
      AND     M1101
      MOV     R1034 D452
      MRD
      AND=    D100 K28
      MOV     R1015 D452
      AND     M152
      AND     M1101
      MOV     R1035 D452
      MRD
      AND=    D100 K30
      MOV     R1016 D452
      AND     M152
      AND     M1101
      MOV     R1036 D452
      MPP
      AND=    D100 K32
      MOV     R1017 D452
      AND     M152
      AND     M1101
      MOV     R1037 D452
